{attribute addProperty BoxType "EJ7342-0000-0019"}
{attribute addProperty Id "ControlAT %Q*Control_E8AFF3DF1620Set_counter_valueAT %Q*UINT16217"}
{attribute addProperty CRC "1552329373"}
{attribute addProperty SizeInBites "32"}
{attribute addProperty SizeInBytes "4"}
TYPE ENC_Control_compact_Channel_5C86AA9D :
STRUCT
	{attribute addProperty Name "Control"}
	Control AT %Q* : Control_E8AFF3DF;
	{attribute addProperty Name "Set_counter_value"}
	Set_counter_value AT %Q* : UINT;
END_STRUCT
END_TYPE

(* stored: Version 1.2.0.0, ProductVersion 3.1.4024.9
   DUT ENC_Control_compact_Channel_5C86AA9D: Id {31066be2-4ea6-4d23-853f-f1229afdc588} *)
